// TIA Portal project "Lab8HMI" (V16)

(* hardware
DEVICE "S71500/ET200MP station_1"  S7-1500 station
   slot 0: "Rail_0"  Rack  6ES7 590-1***0-0AA0
   slot 1: "PLC_1"  CPU 1516-3 PN/DP  6ES7 516-3AN01-0AB0  V2.8
      slot 3: "CPU display_1"  6ES7591-1BA00-0AA0
      slot 32768: "PROFINET interface_1"  X1
         slot 32769: "Port_1"  X1 P1
         slot 32770: "Port_2"  X1 P2
      slot 33024: "PROFINET interface_2"  X2
         slot 33025: "Port_1"  X2 P1
      slot 33280: "DP interface_1"  X3
      slot 34817: "Virtual CP interface port_1"  Virtual CP interface port  Virtual CP interface port
DEVICE "PC station"  SIMATIC PC station
   slot 0: "PC station"  Rail  SIMATIC PC-Station  V1.0
      slot 125: "Stationmanager"  Station_Manager  V6.0.4
   slot 1: "IE general_1"  IE General  IE_CP  V8.2.0
   slot 2: "HMI_RT_1"  WinCC RT Advanced  6AV2 104-0xxxx-xxxx  16.0.0.0
      slot 33792: "Computer interface"  Host interface
*)

// ===== PLC "PLC_1"  CPU 1516-3 PN/DP =====

TYPE "typePIDCompact"
   STRUCT
      setpoint : Real;
      input : Real;
      output : Real;
      state : Int;
      error : Bool;
      distrubOn : Bool;
      errorBits : DWord;
      modeActive : Bool := 1;
      mode : Int := 3;
   END_STRUCT;
END_TYPE

TYPE "typePT3"
   STRUCT
      input : Real;
      tmLag1 : Real := 29.0;
      tmLag2 : Real := 17.5;
      tmLag3 : Real := 3.1;
      gain : Real := 1.0;
      disturb : Real := 0.0;
      cycle : Real := 0.3;
      reset : Bool;
      error : Bool;
      status : Word := 16#0;
      output : Real;
   END_STRUCT;
END_TYPE

DATA_BLOCK "DBTags"   // DB100
{ S7_Optimized_Access := 'TRUE' }
VERSION : 0.1
   VAR
      PIDCompact : "typePIDCompact";
      PT3 : "typePT3";
   END_VAR
BEGIN
END_DATA_BLOCK

DATA_BLOCK "LSim_PT3_DB"   // DB101
{ S7_Optimized_Access := 'TRUE' }
VERSION : 2.01
// stored: InstanceOfName LSim_PT3
"LSim_PT3"
BEGIN
END_DATA_BLOCK

FUNCTION_BLOCK "LSim_PT3"   // FB54, SCL
{ S7_Optimized_Access := 'TRUE' }
VERSION : 2.01
   VAR_INPUT
      input : Real;   // input variable
      tmLag1 : Real := 29.0;   // time lag 1 in s
      tmLag2 : Real := 17.5;   // time lag 2 in s
      tmLag3 : Real := 3.1;   // time lag 3 in s
      gain : Real := 1.0;   // proportional gain
      disturb : Real;   // disturbance variable (additional to "input")
      cycle : Real := 0.1;   // sample time [in sec]
      reset : Bool;   // complete restart (#output = #input)
   END_VAR
   VAR_OUTPUT
      error : Bool;   // error (#tmLag1 <= 0 or #tmLag2 <= 0 or #tmLag3 <= 0)
      status : Word;   // status (if #error = TRUE then status = 16#8001)
      output : Real;   // output signal (if #error = FALSE)
   END_VAR
   VAR
      statFback1 : Real;   // feedback path value 1
      statFback2 : Real;   // feedback path value 2
      statFback3 : Real;   // feedback path value 3
   END_VAR
   VAR_TEMP
      tempHvar : Real;   // help variable
      tempCycleR : Real;   // cycle to real
      tempTmLag1R : Real;   // time lag 1 to real
      tempTmLag2R : Real;   // time lag 2 to real
      tempTmLag3R : Real;   // time lag 3 to real
      tempOutvNew : Real;   // new output variable
   END_VAR
BEGIN
   //=============================================================================
   //SIEMENS AG
   //(c)Copyright 2017 All Rights Reserved
   //-----------------------------------------------------------------------------
   //Library:       Library for Controlled System Simulation
   //Tested with:   S7-1500 FW V2.0 / S7-1200 FW V4.2
   //Engineering:   STEP 7 V14 Upd2 (TIA Portal)
   //Restrictions:  Cyclic interrupt
   //Requirements:  memory card needed for S7-1500
   //Functionality: Simulation of an PT3-system
   //
   //                               gain
   //  F(p) = ------------------------------------------------------
   //         (tmLag1 * p + 1) * (tmLag2 * p + 1) * (tmLag3 * p + 1)
   //          
   //  Call the simulation in a cyclic interrupt with
   //  cyclic interrupt time at least = tmLag1/10!
   //-----------------------------------------------------------------------------
   //Change log table:
   //Version  Date       Expert in charge                Changes applied
   //02.00.00 03.02.2016 Siemens Industry Online Support Release (STEP 7 V13 SP1)
   //02.00.01 02.03.2017 Siemens Industry Online Support Release (STEP 7 V14)
   //=============================================================================
   // check parameter
   IF #tmLag1 <= 0 OR #tmLag2 <= 0 OR #tmLag3 <= 0 THEN
     #error := TRUE;
     #status := W#16#8001;     // Parameter Error
     #output := #input; //write output data
     #statFback1 := #input; //write static data
     #statFback2 := #input;
     #statFback3 := #input;
     RETURN;
   ELSE
     #error := FALSE;
     #status := W#16#0000;     // no error
   END_IF;

   IF #reset THEN //complete restart routine

     #output := #input;//write output data
     #statFback1 := #input;//write static data
     #statFback2 := #input;
     #statFback3 := #input;

   ELSE //cycle mode routine

     #tempCycleR  := #cycle*1000; //transform data type
     #tempTmLag1R := #tmLag1*1000;
     #tempTmLag2R := #tmLag2*1000;
     #tempTmLag3R := #tmLag3*1000;

     IF #tempCycleR * 0.5 > #tempTmLag1R THEN //limit TM_LAG1
       #tempTmLag1R := #tempCycleR * 0.5;
     END_IF;

     IF #tempCycleR * 0.5 > #tempTmLag2R THEN //limit TM_LAG2
       #tempTmLag2R := #tempCycleR * 0.5;
     END_IF;

     IF #tempCycleR * 0.5 > #tempTmLag3R THEN //limit TM_LAG2
       #tempTmLag3R := #tempCycleR * 0.5;
     END_IF;

     //1. first order lag algorithm
     #tempHvar     := #tempCycleR / (#tempTmLag1R * 2.0); 
     #tempHvar     := (#gain * (#input + #disturb) - #statFback1) * #tempHvar / (#tempHvar + 1.0);
     #tempOutvNew  := #tempHvar + #statFback1;
     #statFback1  := #tempHvar * 2.0 + #statFback1;

     //2. first order lag algorithm
     #tempHvar     := #tempCycleR / (#tempTmLag2R * 2.0); 
     #tempHvar     := ((#tempOutvNew - #statFback2) * #tempHvar) / (#tempHvar + 1.0);
     #tempOutvNew  := #tempHvar + #statFback2;
     #statFback2  := #tempHvar * 2.0 + #statFback2;

     //3. first order lag algorithm
     #tempHvar     := #tempCycleR / (#tempTmLag3R * 2.0); 
     #tempHvar     := ((#tempOutvNew - #statFback3) * #tempHvar) / (#tempHvar + 1.0);
     #tempOutvNew  := #tempHvar + #statFback3;
     #statFback3  := #tempHvar * 2.0 + #statFback3;

     #output := #tempOutvNew; //write output

   END_IF;
END_FUNCTION_BLOCK

ORGANIZATION_BLOCK "Main"   // OB1, LAD, ProgramCycle
TITLE = "Main Program Sweep (Cycle)"
{ S7_Optimized_Access := 'TRUE' }
VERSION : 0.1
   VAR_INPUT
      Initial_Call : Bool;   // Initial call of this OB
      Remanence : Bool;   // =True, if remanent data are available
   END_VAR
BEGIN
END_ORGANIZATION_BLOCK

ORGANIZATION_BLOCK "Cyclic interrupt"   // OB30, LAD, CyclicInterrupt
{ S7_Optimized_Access := 'TRUE' }
VERSION : 0.1
   VAR_INPUT
      Initial_Call : Bool;   // Initial call of this OB
      Event_Count : Int;   // Events discarded
   END_VAR
BEGIN

REGION Network 1
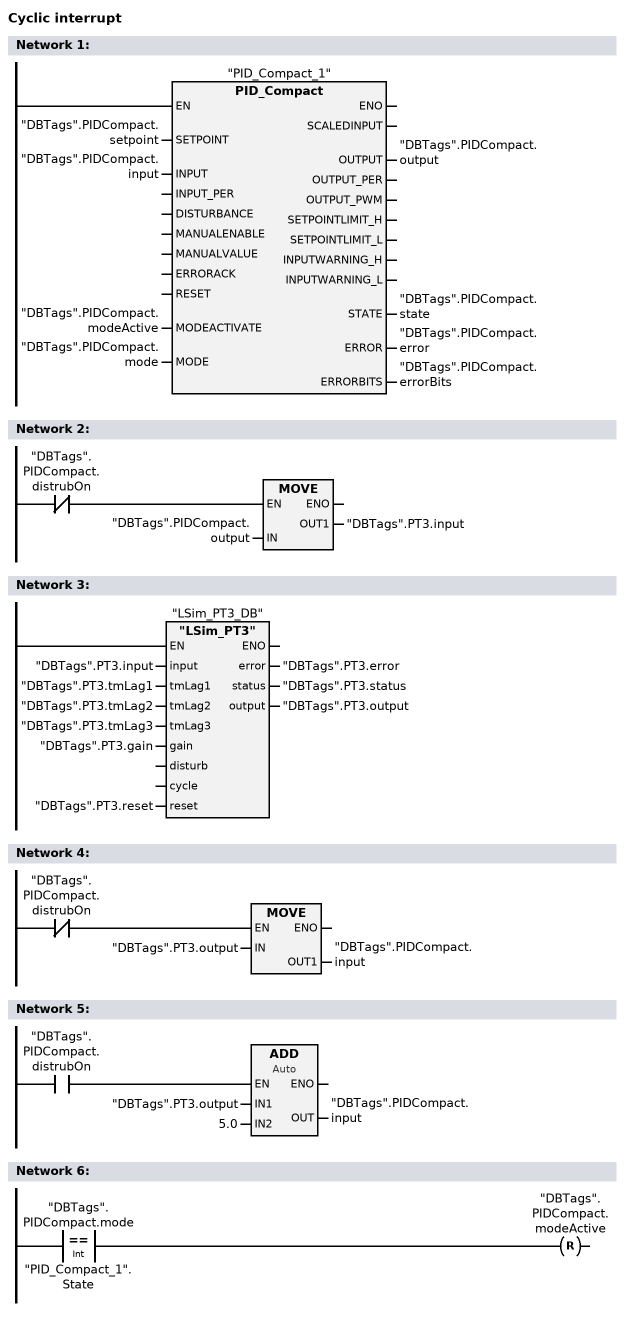
   "PID_Compact_1"(Setpoint := "DBTags".PIDCompact.setpoint,   // PID_Compact
                   Input := "DBTags".PIDCompact.input,
                   ModeActivate := "DBTags".PIDCompact.modeActive,
                   Mode := "DBTags".PIDCompact.mode,
                   Output => "DBTags".PIDCompact.output,
                   State => "DBTags".PIDCompact.state,
                   Error => "DBTags".PIDCompact.error,
                   ErrorBits => "DBTags".PIDCompact.errorBits);
END_REGION

REGION Network 2
   RUNG wire#powerrail
      I_Contact( "DBTags".PIDCompact.distrubOn )
      Move(in := "DBTags".PIDCompact.output, out1 => "DBTags".PT3.input)
   END_RUNG
   // the same network as SCL:
   IF NOT "DBTags".PIDCompact.distrubOn THEN "DBTags".PT3.input := "DBTags".PIDCompact.output; END_IF;
END_REGION

REGION Network 3
   RUNG wire#powerrail
      "LSim_PT3_DB"(input := "DBTags".PT3.input, tmLag1 := "DBTags".PT3.tmLag1, tmLag2 := "DBTags".PT3.tmLag2, tmLag3 := "DBTags".PT3.tmLag3, gain := "DBTags".PT3.gain, disturb :=, cycle :=, reset := "DBTags".PT3.reset, error => "DBTags".PT3.error, status => "DBTags".PT3.status, output => "DBTags".PT3.output)
   END_RUNG
   // the same network as SCL:
   "LSim_PT3_DB"(input := "DBTags".PT3.input,   // "LSim_PT3"
                 tmLag1 := "DBTags".PT3.tmLag1,
                 tmLag2 := "DBTags".PT3.tmLag2,
                 tmLag3 := "DBTags".PT3.tmLag3,
                 gain := "DBTags".PT3.gain,
                 reset := "DBTags".PT3.reset,
                 error => "DBTags".PT3.error,
                 status => "DBTags".PT3.status,
                 output => "DBTags".PT3.output);
END_REGION

REGION Network 4
   RUNG wire#powerrail
      I_Contact( "DBTags".PIDCompact.distrubOn )
      Move(in := "DBTags".PT3.output, out1 => "DBTags".PIDCompact.input)
   END_RUNG
   // the same network as SCL:
   IF NOT "DBTags".PIDCompact.distrubOn THEN "DBTags".PIDCompact.input := "DBTags".PT3.output; END_IF;
END_REGION

REGION Network 5
   RUNG wire#powerrail
      Contact( "DBTags".PIDCompact.distrubOn )
      Add(in1 := "DBTags".PT3.output, in2 := 5.0, out => "DBTags".PIDCompact.input)
   END_RUNG
   // the same network as SCL:
   IF "DBTags".PIDCompact.distrubOn THEN "DBTags".PIDCompact.input := "DBTags".PT3.output + 5.0; END_IF;
END_REGION

REGION Network 6
   RUNG wire#powerrail
      { S7_Templates := "SrcType := Int" } EQ_Contact(in1 := "DBTags".PIDCompact.mode, in2 := "PID_Compact_1".State)
      R_Coil( "DBTags".PIDCompact.modeActive )
   END_RUNG
   // the same network as SCL:
   IF "DBTags".PIDCompact.mode = "PID_Compact_1".State THEN "DBTags".PIDCompact.modeActive := FALSE; END_IF;
END_REGION
END_ORGANIZATION_BLOCK

(* ===== HMI "HMI_RT_1" =====
system functions are stored by id; their names below are inferred from use
connection "HMI_Connection_1": ETHERNET, S7_1500_OMS

HMI tags "Default tag table"
   "PID_Compact_1_RunModeByStartup" : Bool = PLC PID_Compact_1.RunModeByStartup, 1 s
   "PID_Compact_1_Retain_CtrlParams_Td" : Real = PLC PID_Compact_1.Retain.CtrlParams.Td, 1 s
   "PID_Compact_1_Retain_CtrlParams_DWeighting" : Real = PLC PID_Compact_1.Retain.CtrlParams.DWeighting, 1 s
   "PID_Compact_1_Retain_CtrlParams_TdFiltRatio" : Real = PLC PID_Compact_1.Retain.CtrlParams.TdFiltRatio, 1 s
   "PID_Compact_1_Config_InputScaling_UpperPointIn" : Real = PLC PID_Compact_1.Config.InputScaling.UpperPointIn, 1 s
   "PID_Compact_1_Config_InputScaling_LowerPointIn" : Real = PLC PID_Compact_1.Config.InputScaling.LowerPointIn, 1 s
   "PID_Compact_1_Retain_CtrlParams_Ti" : Real = PLC PID_Compact_1.Retain.CtrlParams.Ti, 1 s
   "PID_Compact_1_Config_InvertControl" : Bool = PLC PID_Compact_1.Config.InvertControl, 1 s
   "PID_Compact_1_Config_MinimumOffTime" : Real = PLC PID_Compact_1.Config.MinimumOffTime, 1 s
   "PID_Compact_1_Config_MinimumOnTime" : Real = PLC PID_Compact_1.Config.MinimumOnTime, 1 s
   "PID_Compact_1_Config_OutputUpperLimit" : Real = PLC PID_Compact_1.Config.OutputUpperLimit, 1 s
   "PID_Compact_1_Config_OutputLowerLimit" : Real = PLC PID_Compact_1.Config.OutputLowerLimit, 1 s
   "PID_Compact_1_PhysicalQuantity" : Int = PLC PID_Compact_1.PhysicalQuantity, 1 s
   "PID_Compact_1_Config_InputUpperLimit" : Real = PLC PID_Compact_1.Config.InputUpperLimit, 1 s
   "PID_Compact_1_Config_InputLowerLimit" : Real = PLC PID_Compact_1.Config.InputLowerLimit, 1 s
   "PID_Compact_1_Retain_CtrlParams_PWeighting" : Real = PLC PID_Compact_1.Retain.CtrlParams.PWeighting, 1 s
   "PID_Compact_1_Retain_CtrlParams_Gain" : Real = PLC PID_Compact_1.Retain.CtrlParams.Gain, 1 s
   "PID_Compact_1_Retain_CtrlParams_Cycle" : Real = PLC PID_Compact_1.Retain.CtrlParams.Cycle, 1 s
   "PID_Compact_1_Config_InputScaling_UpperPointOut" : Real = PLC PID_Compact_1.Config.InputScaling.UpperPointOut, 1 s
   "PID_Compact_1_Config_InputScaling_LowerPointOut" : Real = PLC PID_Compact_1.Config.InputScaling.LowerPointOut, 1 s
   "PID_Compact_1_Config_InputPerOn" : Bool = PLC PID_Compact_1.Config.InputPerOn, 1 s
   "PID_Compact_1_Mode" : Int = PLC PID_Compact_1.Mode, 1 s
   "PID_Compact_1_SubstituteOutput" : Real = PLC PID_Compact_1.SubstituteOutput, 1 s
   "PID_Compact_1_PhysicalUnit" : Int = PLC PID_Compact_1.PhysicalUnit, 1 s
   "PID_Compact_1_Config_InputUpperWarning" : Real = PLC PID_Compact_1.Config.InputUpperWarning, 1 s
   "PID_Compact_1_Config_InputLowerWarning" : Real = PLC PID_Compact_1.Config.InputLowerWarning, 1 s
   "PID_Compact_1_CtrlParamsBackUp_Gain" : Real = PLC PID_Compact_1.CtrlParamsBackUp.Gain, 1 s
   "PID_Compact_1_CtrlParamsBackUp_Ti" : Real = PLC PID_Compact_1.CtrlParamsBackUp.Ti, 1 s
   "PID_Compact_1_CtrlParamsBackUp_Td" : Real = PLC PID_Compact_1.CtrlParamsBackUp.Td, 1 s
   "PID_Compact_1_CtrlParamsBackUp_TdFiltRatio" : Real = PLC PID_Compact_1.CtrlParamsBackUp.TdFiltRatio, 1 s
   "PID_Compact_1_CtrlParamsBackUp_PWeighting" : Real = PLC PID_Compact_1.CtrlParamsBackUp.PWeighting, 1 s
   "PID_Compact_1_CtrlParamsBackUp_DWeighting" : Real = PLC PID_Compact_1.CtrlParamsBackUp.DWeighting, 1 s
   "PID_Compact_1_CtrlParamsBackUp_Cycle" : Real = PLC PID_Compact_1.CtrlParamsBackUp.Cycle, 1 s
   "PID_Compact_1_ActivateRecoverMode" : Bool = PLC PID_Compact_1.ActivateRecoverMode, 1 s
   "PID_Compact_1_SetSubstituteOutput" : Bool = PLC PID_Compact_1.SetSubstituteOutput, 1 s
   "PID_Compact_1_PIDSelfTune_SUT_TuneRule" : Int = PLC PID_Compact_1.PIDSelfTune.SUT.TuneRule, 1 s
   "PID_Compact_1_PIDSelfTune_TIR_TuneRule" : Int = PLC PID_Compact_1.PIDSelfTune.TIR.TuneRule, 1 s
   "PID_Compact_1_Setpoint" : Real = PLC PID_Compact_1.Setpoint, 1 s
   "PID_Compact_1_Input" : Real = PLC PID_Compact_1.Input, 1 s
   "PID_Compact_1_Input_PER" : Int = PLC PID_Compact_1.Input_PER, 1 s
   "PID_Compact_1_Disturbance" : Real = PLC PID_Compact_1.Disturbance, 1 s
   "PID_Compact_1_ManualEnable" : Bool = PLC PID_Compact_1.ManualEnable, 1 s
   "PID_Compact_1_ManualValue" : Real = PLC PID_Compact_1.ManualValue, 1 s
   "PID_Compact_1_ErrorAck" : Bool = PLC PID_Compact_1.ErrorAck, 1 s
   "PID_Compact_1_Reset" : Bool = PLC PID_Compact_1.Reset, 1 s
   "PID_Compact_1_ModeActivate" : Bool = PLC PID_Compact_1.ModeActivate, 1 s
   "PID_Compact_1_ScaledInput" : Real = PLC PID_Compact_1.ScaledInput, 1 s
   "PID_Compact_1_Output" : Real = PLC PID_Compact_1.Output, 1 s
   "PID_Compact_1_Output_PER" : Int = PLC PID_Compact_1.Output_PER, 1 s
   "PID_Compact_1_Output_PWM" : Bool = PLC PID_Compact_1.Output_PWM, 1 s
   "PID_Compact_1_SetpointLimit_H" : Bool = PLC PID_Compact_1.SetpointLimit_H, 1 s
   "PID_Compact_1_SetpointLimit_L" : Bool = PLC PID_Compact_1.SetpointLimit_L, 1 s
   "PID_Compact_1_InputWarning_H" : Bool = PLC PID_Compact_1.InputWarning_H, 1 s
   "PID_Compact_1_InputWarning_L" : Bool = PLC PID_Compact_1.InputWarning_L, 1 s
   "PID_Compact_1_State" : Int = PLC PID_Compact_1.State, 1 s
   "PID_Compact_1_Error" : Bool = PLC PID_Compact_1.Error, 1 s
   "PID_Compact_1_ErrorBits" : DWord = PLC PID_Compact_1.ErrorBits, 1 s
   "PID_Compact_1_InternalVersion" : DWord = PLC PID_Compact_1.InternalVersion, 1 s
   "PID_Compact_1_IntegralResetMode" : Int = PLC PID_Compact_1.IntegralResetMode, 1 s
   "PID_Compact_1_OverwriteInitialOutputValue" : Real = PLC PID_Compact_1.OverwriteInitialOutputValue, 1 s
   "PID_Compact_1_LoadBackUp" : Bool = PLC PID_Compact_1.LoadBackUp, 1 s
   "PID_Compact_1_Warning" : DWord = PLC PID_Compact_1.Warning, 1 s
   "PID_Compact_1_WarningInternal" : DWord = PLC PID_Compact_1.WarningInternal, 1 s
   "PID_Compact_1_Progress" : Real = PLC PID_Compact_1.Progress, 1 s
   "PID_Compact_1_CurrentSetpoint" : Real = PLC PID_Compact_1.CurrentSetpoint, 1 s
   "PID_Compact_1_CancelTuningLevel" : Real = PLC PID_Compact_1.CancelTuningLevel, 1 s
   "PID_Compact_1_Config_SetpointUpperLimit" : Real = PLC PID_Compact_1.Config.SetpointUpperLimit, 1 s
   "PID_Compact_1_Config_SetpointLowerLimit" : Real = PLC PID_Compact_1.Config.SetpointLowerLimit, 1 s
   "PID_Compact_1_CycleTime_StartEstimation" : Bool = PLC PID_Compact_1.CycleTime.StartEstimation, 1 s
   "PID_Compact_1_CycleTime_EnEstimation" : Bool = PLC PID_Compact_1.CycleTime.EnEstimation, 1 s
   "PID_Compact_1_CycleTime_EnMonitoring" : Bool = PLC PID_Compact_1.CycleTime.EnMonitoring, 1 s
   "PID_Compact_1_CycleTime_Value" : Real = PLC PID_Compact_1.CycleTime.Value, 1 s
   "PID_Compact_1_PIDSelfTune_SUT_CalculateParams" : Bool = PLC PID_Compact_1.PIDSelfTune.SUT.CalculateParams, 1 s
   "PID_Compact_1_PIDSelfTune_SUT_State" : Int = PLC PID_Compact_1.PIDSelfTune.SUT.State, 1 s
   "PID_Compact_1_PIDSelfTune_TIR_RunIn" : Bool = PLC PID_Compact_1.PIDSelfTune.TIR.RunIn, 1 s
   "PID_Compact_1_PIDSelfTune_TIR_CalculateParams" : Bool = PLC PID_Compact_1.PIDSelfTune.TIR.CalculateParams, 1 s
   "PID_Compact_1_PIDSelfTune_TIR_State" : Int = PLC PID_Compact_1.PIDSelfTune.TIR.State, 1 s
   "PID_Compact_1_PIDCtrl_PIDInit" : Bool = PLC PID_Compact_1.PIDCtrl.PIDInit, 1 s
   "PID_Compact_1_PIDCtrl_IntegralSum" : Real = PLC PID_Compact_1.PIDCtrl.IntegralSum, 1 s
   "DBTags_PIDCompact_setpoint" : Real = PLC DBTags.PIDCompact.setpoint AT %DB1.DBD0, 1 s
   "DBTags_PIDCompact_input" : Real = PLC DBTags.PIDCompact.input AT %DB1.DBD0, 1 s
   "DBTags_PIDCompact_output" : Real = PLC DBTags.PIDCompact.output AT %DB1.DBD0, 1 s
   "DBTags_PIDCompact_state" : Int = PLC DBTags.PIDCompact.state AT %DB1.DBD0, 1 s
   "DBTags_PIDCompact_error" : Bool = PLC DBTags.PIDCompact.error AT %DB1.DBD0, 1 s
   "DBTags_PIDCompact_distrubOn" : Bool = PLC DBTags.PIDCompact.distrubOn AT %DB1.DBD0, 1 s
   "DBTags_PIDCompact_errorBits" : DWord = PLC DBTags.PIDCompact.errorBits AT %DB1.DBD0, 1 s
   "DBTags_PIDCompact_modeActive" : Bool = PLC DBTags.PIDCompact.modeActive AT %DB1.DBD0, 1 s
   "DBTags_PIDCompact_mode" : Int = PLC DBTags.PIDCompact.mode AT %DB1.DBD0, 1 s
   "DBTags_PT3_tmLag1" : Real = PLC DBTags.PT3.tmLag1, 1 s
   "DBTags_PT3_tmLag2" : Real = PLC DBTags.PT3.tmLag2, 1 s

screen "PIDTest" 1024x768
   Button "Button_1" at 104,33 size 111x31; TextOff 'Stop Run Time'
      on Release: StopRuntime(0)
      on Click: StopRuntime(0)
   TextField "Text field_1" at 14,2 size 297x22; Text 'Automation Technoglogy Lab session 7'
   Button "Button_2" at 122,224 size 85x31; TextOff 'PID Test'
      on Release: ActivateScreen("PIDTest", 0)
   TrendView "Trend view_1" at 207,18 size 733x357
   IOField "I/O field_1" at 72,72 size 130x32; FormatPattern s999.999
      ProcessValue <- "PID_Compact_1_Retain_CtrlParams_Gain"
   TextField "Text field_2" at 14,82 size 39x22; Text 'Gain'
   IOField "I/O field_2" at 74,112 size 130x33; FormatPattern s999.999
      ProcessValue <- "PID_Compact_1_Retain_CtrlParams_Ti"
   IOField "I/O field_3" at 76,158 size 129x33; FormatPattern s999.999
      ProcessValue <- "PID_Compact_1_Retain_CtrlParams_Td"
   TextField "Text field_3" at 23,119 size 19x22; Text 'Ti'
   TextField "Text field_4" at 23,161 size 23x22; Text 'Td'
   Switch "Switch_1" at 46,287 size 134x53; CaptionText 'Switch'; TextOff 'OFF'; TextOn 'ON'
      ProcessValue <- "DBTags_PIDCompact_distrubOn"
   Button "Button_3" at 34,357 size 142x44; TextOff 'Auto mode'
      on Press: SetTag("DBTags_PIDCompact_mode", 3)
      on Release: SetBit("DBTags_PIDCompact_modeActive")
      Appearance <- "DBTags_PIDCompact_mode"
   Button "Button_4" at 34,414 size 142x44; TextOff 'Manual mode'
      on Release: SetBit("DBTags_PIDCompact_modeActive")
      Appearance <- "DBTags_PIDCompact_mode"
      on Press: SetTag("DBTags_PIDCompact_mode", 4)
   IOField "I/O field_4" at 206,405 size 123x32; FormatPattern s999.999
      ProcessValue <- "DBTags_PIDCompact_setpoint"
   TextField "Text field_5" at 206,368 size 73x22; Text 'Set Point'
   IOField "I/O field_5" at 206,462 size 123x32; FormatPattern s999.999
      ProcessValue <- "PID_Compact_1_ManualValue"
   TextField "Text field_6" at 203,499 size 194x22; Text 'Controller Manual Output'
   IOField "I/O field_6" at 630,414 size 106x32; FormatPattern s999.999
      ProcessValue <- "DBTags_PIDCompact_output"
   TextField "Text field_7" at 627,393 size 136x22; Text 'Controller Output'
   IOField "I/O field_7" at 869,414 size 106x32; FormatPattern s999.999
      ProcessValue <- "DBTags_PIDCompact_input"
   TextField "Text field_8" at 841,379 size 167x22; Text 'Process value (Input)'
   Button "Button_5" at 6,33 size 96x32; TextOff 'Start'
      on Release: ActivateScreen("Start", 0)
   IOField "I/O field_8" at 32,499 size 123x32; FormatPattern s999999999.999
      ProcessValue <- "DBTags_PT3_tmLag1"
   TextField "Text field_9" at 34,472 size 57x22; Text 'tmlag1'
   IOField "I/O field_9" at 34,538 size 123x32; FormatPattern s999999999.999
      ProcessValue <- "DBTags_PT3_tmLag2"
   IOField "I/O field_10" at 36,577 size 123x32; FormatPattern s999999999.999
      ProcessValue <- "DBTags_PT3_tmLag1"

screen "Start" 1024x768
   TextField "Text field_1" at 123,73 size 286x22; Text 'Automation Technology Lab Session 7'
   Button "Button_1" at 165,115 size 153x59; TextOff 'PID Test'
      on Release: ActivateScreen("PIDTest", 0)
   Button "Button_2" at 535,120 size 170x51; TextOff 'Stop Runtime'
      on Click: StopRuntime(0)
   GraphicView "Graphic view_1" at 403,119 size 58x58; Picture "Graphic_2"
   GraphicView "Graphic view_2" at 535,14 size 158x106; Picture "Graphic_3"
*)